FUNCTION_BLOCK FB_PWM
VAR_INPUT
	SafeetyOk : BOOL;
	Torque: INT;
END_VAR

VAR
  	ModuleState AT %I* : UINT;
	
 	Control AT %Q* :  UINT;
 	TargetTorque AT %Q*: INT; 	

 	State  : INT := 1;
 	PwmTimer : ton;
END_VAR



CASE State OF 

	1:
		IF SafeetyOk THEN
			State := 2;
		END_IF
	2: 
		Control := 6;
		IF ModuleState = 40 OR ModuleState = 33 THEN
			State := 5;
		END_IF
	5:
		Control := 128;
		IF ModuleState = 96 OR ModuleState = 33 OR ModuleState = 168 THEN
			State := 10;
		END_IF
	10:
		Control := 6;
		IF ModuleState = 33 THEN
			state := 15;
		END_IF	
	15:
		Control := 7;
		IF ModuleState = 35 OR ModuleState = 163 or ModuleState = 2083 THEN
			State := 20;
		END_IF	
	20:	
		Control := 15;
		IF ModuleState = 4135 OR ModuleState = 4263THEN
			state := 25;
		END_IF
	24:
	  //IF Torque = 0  THEN
			State := 25;
	//	END_IF	
		PwmTimer(in := FALSE,PT := T#30S);
	25:
		IF ModuleState = 40 THEN
			State := 5;
		END_IF
		
		IF Torque > 0 THEN
			TargetTorque := Torque ;
		ELSIF Torque = 0 AND TargetTorque > 0  THEN	
			TargetTorque :=  TargetTorque - REAL_TO_INT((INT_TO_REAL(TargetTorque)*0.07));
		END_IF	
		
		PwmTimer(in := TargetTorque > 300,PT := T#30S);
		IF PwmTimer.Q  THEN
			PwmTimer(in := FALSE,PT := T#30S);
			State := 35;
		END_IF 
	35:
		IF TargetTorque >0 THEN
			TargetTorque := TargetTorque -4;
		ELSIF 	TargetTorque = 0  THEN
				State := 24;
		END_IF	

END_CASE

END_FUNCTION_BLOCK

(* stored: Version 1.1.0.1, ProductVersion 3.1.4026.8
   POU FB_PWM: Id {09b123ef-3dc6-4859-9f9a-c8c3fdb58c25}, SpecialFunc None *)
